{attribute 'GeneratedUsingTerminal: EL2014-0000-0016'}
{attribute addProperty BoxType "EL2014-0000-0016"}
{attribute addProperty Id "AdsAddrAT %I*.TcoAmsAddr0StateAT %I*UINT2"}
{attribute addProperty CRC "2493615966"}
{attribute addProperty Size "2"}
TYPE InfoData_94A18F5E :
STRUCT
	{attribute addProperty Name "AdsAddr"}
	AdsAddr AT %I* : .TcoAmsAddr;
	{attribute addProperty Name "State"}
	State AT %I* : UINT;
END_STRUCT
END_TYPE

(* stored: Version 1.2.0.0, ProductVersion 3.1.4024.9
   DUT InfoData_94A18F5E: Id {eb41a35d-a852-44d9-a4f3-cd6759847859} *)
